{attribute 'GeneratedUsingTerminal: EL2014-0000-0017'}
{attribute addProperty BoxType "EL2014-0000-0017"}
{attribute addProperty Id "EtcSlaveTerminalBaseDIG_OutputsAT %Q*DIG_Outputs_F9744C664WcStateAT %I*WcState_0B2B16F91InfoDataAT %I*InfoData_32EB74EA10"}
{attribute addProperty CRC "4161326580"}
{attribute addProperty Size "15"}
TYPE EL2014_F808CDF4 EXTENDS EtcSlaveTerminalBase :
STRUCT
	{attribute addProperty Name "DIG_Outputs"}
	DIG_Outputs : DIG_Outputs_F9744C66;
	{attribute addProperty Name "WcState"}
	WcState : WcState_0B2B16F9;
	{attribute addProperty Name "InfoData"}
	InfoData : InfoData_32EB74EA;
END_STRUCT
END_TYPE

(* stored: Version 1.2.0.0, ProductVersion 3.1.4024.9
   DUT EL2014_F808CDF4: Id {120b29fa-c3ef-4e27-97b1-e5ba2848389d} *)
